# EPICS StreamDevice protocol: protocols/k2461.proto
Terminator = CR LF;

setCurrLim {
    out "SOUR:VOLT:ILIM %.2f";
}
